FUNCTION_BLOCK PUBLIC StationManager
VAR_INPUT
END_VAR
VAR_OUTPUT
END_VAR
VAR
END_VAR

;

METHOD PUBLIC NotifyStationNewVehArrival : BOOL
VAR_INPUT
	Pos 			:	REAL;
	StationIndex 	:	BYTE;
	VehicleID		:	BYTE;
END_VAR
CASE StationIndex OF

 
MM_CONST.LOAD_1_STA:
	Stations.fbLoad1Sta.VehicleUnderTest := VehicleID;	
    Stations.fbLoad1Sta.Trigger := TRUE;
		

MM_CONST.LOAD_2_STA:
	Stations.fbLoad2Sta.VehicleUnderTest := VehicleID;		   
    Stations.fbLoad2Sta.Trigger := TRUE;
        			
MM_CONST.LOAD_3_STA:
	Stations.fbLoad3Sta.VehicleUnderTest := VehicleID;	
	Stations.fbLoad3Sta.Trigger := TRUE;					

MM_CONST.LOAD_4_STA:					
	Stations.fbLoad4Sta.VehicleUnderTest := VehicleID;
	Stations.fbLoad4Sta.Trigger := TRUE;	

MM_CONST.STOP_BEFORE_VISION_STA:
	Stations.fbOB_StopBeforeVisionSta.VehicleUnderTest := VehicleID;
	Stations.fbOB_StopBeforeVisionSta.Trigger := TRUE;

MM_CONST.VISION_STA:
	Stations.fbVisionSta.VehicleUnderTest := VehicleID;
	Stations.fbVisionSta.Trigger := TRUE;

MM_CONST.PISTON_STA:
	Stations.fbPistonSta.VehicleUnderTest := VehicleID;
	Stations.fbPistonSta.Trigger := TRUE;

MM_CONST.CAP_STA:
	Stations.fbCapInsertSta.VehicleUnderTest := VehicleID;
	Stations.fbCapInsertSta.Trigger := TRUE;

MM_CONST.IB_STOP_ROBOT_CLEAR_STA:
	Stations.fbIB_StopRobotSta.VehicleUnderTest := VehicleID;
	Stations.fbIB_StopRobotSta.Trigger := TRUE;

MM_CONST.REJECT_ULOAD_STA:
	Stations.fbRejectSta.VehicleUnderTest := VehicleID;
	Stations.fbRejectSta.Trigger := TRUE;

MM_CONST.GOOD_UL_1_STA:
	Stations.fbGoodULSta_1.VehicleUnderTest := VehicleID;
	Stations.fbGoodULSta_1.Trigger := TRUE;

MM_CONST.GOOD_UL_2_STA:
	Stations.fbGoodULSta_2.VehicleUnderTest := VehicleID;
	Stations.fbGoodULSta_2.Trigger := TRUE;

MM_CONST.GOOD_UL_3_STA:
	Stations.fbGoodULSta_3.VehicleUnderTest := VehicleID;
	Stations.fbGoodULSta_3.Trigger := TRUE;

MM_CONST.GOOD_UL_4_STA:
	Stations.fbGoodULSta_4.VehicleUnderTest := VehicleID;
	Stations.fbGoodULSta_4.Trigger := TRUE;

(*	
MM_CONST.GOOD_UNLOAD_STA:
	Stations.fbGoodUnloadSta.VehicleUnderTest := VehicleID;
	Stations.fbGoodUnloadSta.Trigger := TRUE;	
 *)   
MM_CONST.OB_STOP_ROBOT_CLEAR_STA:
	Stations.fbOB_StopRobotSta.VehicleUnderTest := VehicleID;  
    Stations.fbOB_StopRobotSta.Trigger := TRUE;
ELSE ;
	
END_CASE
END_METHOD

END_FUNCTION_BLOCK

(* stored: Version 1.1.0.1, ProductVersion 3.1.4022.6
   POU StationManager: Id {3bea6e74-ad93-4a06-afc2-89b8f54cda95}, SpecialFunc None
   Method NotifyStationNewVehArrival: Id {ea3af994-aee1-46c5-a0f2-3db7a4ef7bf1} *)
